Universal Robots PolyScope program: minipjoan.urp

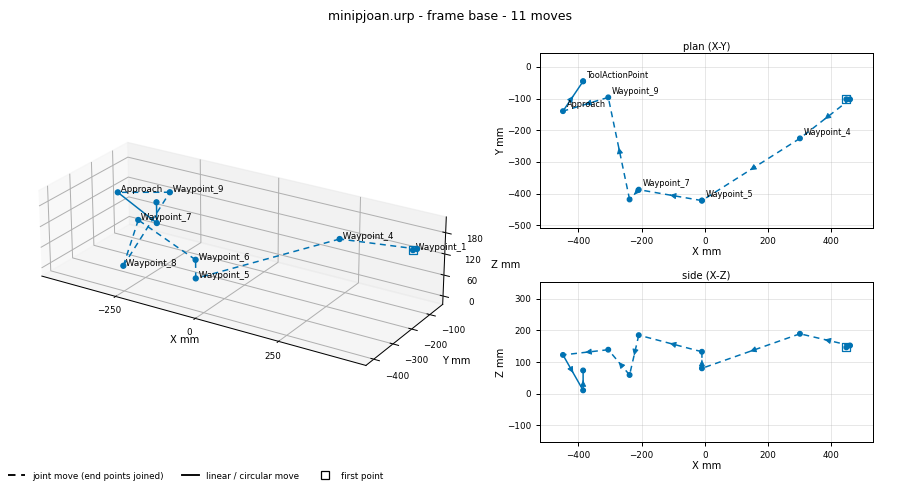
[picture p0: tool path of minipjoan.urp in frame base, 11 of 12 moves have a stored position in this frame; points joined in program order, loops and branches not executed]
Program minipjoan (installation=default directory=/programs createdIn=5.14.5 lastSavedIn=5.14.5 robotSerialNumber=20195300809)
Calibrated DH parameters: a=[-0.000085, -0.20076, -0.212369, 0.000121, -0.000118, 0]; d=[0.15185, -26.306375, 24.753047, 1.684739, 0.085386, 0.092088]; alpha=[1.572149, -0.00522, -0.011864, 1.571339, -1.571085, 0]; deltaTheta=[0, 0.599885, -0.513355, -0.086555, 0.000006, 0]
InitVariablesNode variables(variable(name=Pallet_1_cnt_1, expression=1), variable(name=Pallet_1_lct, expression=1), variable(name=Pallet_1_lno, expression=1), variable(name=Pallet_1_sep, expression=False), variable(name=Pallet_1_tct, expression=1))
Robot Program (runOnlyOnce=false)
  URCap Gripper Activate (Robotiq_Grippers, Robotiq Inc.) dataModel(ResetAndActivateKey=false)
  MoveJ speed 60 deg/s, acceleration 80 deg/s^2 (useActiveTCP=true) feature=Base
    Waypoint Waypoint_1: TCP in base x=447.267 y=-102.061 z=146.421 mm, rx=-2.205 ry=2.174 rz=-0.1317 rad; joints [4.81, -119.207, -49.648, -96.135, 87.137, 4.36] deg; TCP offset x=0 y=0 z=174 mm, rx=0 ry=0 rz=0 rad
  URCap Gripper (Robotiq_Grippers, Robotiq Inc.) dataModel(position=100.0, force=0.0, speed=0.0, positionInDouble=100.0, forceInDouble=0.0, speedInDouble=0.0, slaveIds=[9], blocking=true)
  MoveL speed 250 mm/s, acceleration 1200 mm/s^2 (useActiveTCP=true) feature=Base
    MoveDirectionNode (selectedDirection=ZMinus toolParams=0.05, 1.2)
      Until TOOL_CONTACT_DETECTION (allowActions=true retraction=0.005 decelerationAcceleration=3 decelerationAngularAcceleration=34.906585)
        URCap Gripper (Robotiq_Grippers, Robotiq Inc.) dataModel(position=0.0, force=0.0, speed=0.0, positionInDouble=0.0, forceInDouble=0.0, speedInDouble=0.0, slaveIds=[9], blocking=true)
        MoveL speed 250 mm/s, acceleration 1200 mm/s^2 (useActiveTCP=true) feature=Base
          Waypoint Waypoint_2 (Relative): relativeFromPosition TCP in base x=471.213 y=-99.416 z=63.282 mm, rx=-2.1249 ry=2.1283 rz=-0.2138 rad; joints [4.58, -119.887, -74.402, -64.902, 87.774, 4.609] deg; TCP in base x=479.804 y=-96.799 z=39.969 mm, rx=-2.142 ry=2.1284 rz=-0.2147 rad; joints [5.105, -123.73, -74.341, -61.658, 87.263, 4.605] deg
          URCap Gripper (Robotiq_Grippers, Robotiq Inc.) dataModel(position=58.431372549019606, force=0.0, speed=0.0, positionInDouble=58.431372549019606, forceInDouble=0.0, speedInDouble=0.0, slaveIds=[9], blocking=true)
          Waypoint Waypoint_3: TCP in base x=458.907 y=-102.285 z=152.325 mm, rx=-2.0281 ry=2.0188 rz=-0.3366 rad; joints [3.504, -105.987, -77.03, -66.932, 89.229, 3.326] deg
  MoveJ speed 60 deg/s, acceleration 80 deg/s^2 (useActiveTCP=true) feature=Base
    Waypoint Waypoint_4: TCP in base x=300.574 y=-225.676 z=189.373 mm, rx=-0.8393 ry=3.0246 rz=-0.1221 rad; joints [-13.828, -100.697, -62.451, -104.67, 85.518, 45.615] deg
    MoveJ speed 60 deg/s, acceleration 80 deg/s^2 (useActiveTCP=true) feature=Base
      Waypoint Waypoint_5: TCP in base x=-9.268 y=-422.356 z=80.192 mm, rx=-0.0596 ry=3.0948 rz=-0.085 rad; joints [-74.508, -112.122, -77.499, -76.664, 91.009, 13.565] deg
      URCap Gripper (Robotiq_Grippers, Robotiq Inc.) dataModel(position=0.0, force=0.0, speed=0.0, positionInDouble=0.0, forceInDouble=0.0, speedInDouble=0.0, slaveIds=[9], blocking=true)
      MoveJ speed 60 deg/s, acceleration 80 deg/s^2 (useActiveTCP=true) feature=Base
        Waypoint Waypoint_6: TCP in base x=-9.251 y=-422.355 z=132.542 mm, rx=-0.0597 ry=3.0948 rz=-0.085 rad; joints [-74.543, -111.435, -64.364, -90.485, 91.014, 13.69] deg
        Wait Sleep waitTime=8
    MoveJ speed 60 deg/s, acceleration 80 deg/s^2 (useActiveTCP=true) feature=Base
      Waypoint Waypoint_7: TCP in base x=-208.935 y=-387.816 z=185.052 mm, rx=0.0938 ry=-3.0517 rz=0.1155 rad; joints [44.36, -64.936, 47.012, -78.661, -91.033, -48.996] deg
      MoveJ speed 60 deg/s, acceleration 80 deg/s^2 (useActiveTCP=true) feature=Base
        Waypoint Waypoint_8: TCP in base x=-237.941 y=-418.796 z=59.161 mm, rx=0.0915 ry=-3.1228 rz=-0.0431 rad; joints [45.6, -46.032, 46.886, -90.484, -92.713, -47.784] deg
        URCap Gripper (Robotiq_Grippers, Robotiq Inc.) dataModel(position=58.03921568627451, force=0.0, speed=0.0, positionInDouble=58.03921568627451, forceInDouble=0.0, speedInDouble=0.0, slaveIds=[9], blocking=true)
      MoveJ speed 60 deg/s, acceleration 80 deg/s^2 (useActiveTCP=true) feature=Base
        Waypoint Waypoint_9: TCP in base x=-305.318 y=-96.059 z=139.035 mm, rx=-2.0283 ry=-2.295 rz=0.0831 rad; joints [-7.04, -97.483, 97.145, -95.102, -90.705, -13.988] deg
        URCap Palletizing (polyscope-pallet-impl, Universal Robots) dataModel(palletFeature=Base, isPalletizing=true, Variable(key=name, variable(name=Pallet_1)), Variable(key=globalCountingVariable, variable(name=Pallet_1_cnt_1, initializeExpression=1)), Variable(key=layerNumberVariable, variable(name=Pallet_1_lno, initializeExpression=1)), Variable(key=layerCountingVariable, variable(name=Pallet_1_lct, initializeExpression=1)), Variable(key=handleSeparatorVariable, variable(name=Pallet_1_sep, initializeExpression=False)), Variable(key=totalCountVariable, variable(name=Pallet_1_tct, initializeExpression=1)), Variable(key=referencePoint, variable(featureName=referencePoint)), Variable(key=separatorPoint, variable(featureName=separatorPoint)), Length(key=objectHeight value=0.04 unit=M)); state(isChildrenLocked=true)
          URCap Patterns (polyscope-pallet-impl, Universal Robots) state(isChildrenLocked=true)
            URCap Pattern (polyscope-pallet-impl, Universal Robots) dataModel(UUID=86fc2707-347a-4276-997c-d25539b2d56b, patternType=GRID, rows=3, columns=4, Variable(key=nameVariable, variable(name=Grid_Pattern_1))); state(isChildrenLocked=true)
              URCap Item (polyscope-pallet-impl, Universal Robots) dataModel(UUID=84c2eab7-4ccd-47c8-9968-c744c75cb5a4, patternType=GRID, index=0, calibrationDeltaTheta=[2.0871938292282843E-8, 0.5998849625986696, -0.513354759222901, -0.08655474087847535, 6.239817607139875E-6, -6.658617090343766E-8], calibrationA=[-8.52060452638757E-5, -0.2007601879611388, -0.2123691625519033, 1.2105607098011576E-4, -1.1833705743435544E-4, 0.0], calibrationD=[0.15184970286177432, -26.306374840159272, 24.75304670983349, 1.6847390881089916, 0.085385969004481, 0.09208826337351553], calibrationAlpha=[1.5721487795181908, -0.005219907129425837, -0.011864150755780208, 1.5713392161993658, -1.5710853432049288, 0.0], calibrationJointChecksum=[-1860213401, -1859864814, -1494669377, -1328152407, -1329437658, -1329056899], calibrationStatus=2, calibrationValidChecksum=true, baseToFeature=[0.0, 0.0, 0.0, 0.0, 0.0, 0.0], TCPOffset=[-4.9798563925285144E-8, -1.1903855710371225E-5, 0.17398545185544173, 3.862269624087422E-5, 1.2921357085209562E-5, -2.2884874203884517E-5], Variable(key=variable, variable(name=CornerItem_1)), JointPositions(key=jointpositions, JointPosition(key=[1], Angle(key=pos value=-0.188365 unit=RAD)), JointPosition(key=[2], Angle(key=pos value=-1.19048 unit=RAD)), JointPosition(key=[3], Angle(key=pos value=1.760904 unit=RAD)), JointPosition(key=[4], Angle(key=pos value=-2.274609 unit=RAD)), JointPosition(key=[5], Angle(key=pos value=-1.616725 unit=RAD)), JointPosition(key=[6], Angle(key=pos value=-0.207331 unit=RAD))))
              URCap Item (polyscope-pallet-impl, Universal Robots) dataModel(UUID=72bba91b-081b-49f2-b649-66cb13c50b99, patternType=GRID, index=1, calibrationDeltaTheta=[2.0871938292282843E-8, 0.5998849625986696, -0.513354759222901, -0.08655474087847535, 6.239817607139875E-6, -6.658617090343766E-8], calibrationA=[-8.52060452638757E-5, -0.2007601879611388, -0.2123691625519033, 1.2105607098011576E-4, -1.1833705743435544E-4, 0.0], calibrationD=[0.15184970286177432, -26.306374840159272, 24.75304670983349, 1.6847390881089916, 0.085385969004481, 0.09208826337351553], calibrationAlpha=[1.5721487795181908, -0.005219907129425837, -0.011864150755780208, 1.5713392161993658, -1.5710853432049288, 0.0], calibrationJointChecksum=[-1860213401, -1859864814, -1494669377, -1328152407, -1329437658, -1329056899], calibrationStatus=2, calibrationValidChecksum=true, baseToFeature=[0.0, 0.0, 0.0, 0.0, 0.0, 0.0], TCPOffset=[1.7947581433003235E-5, -3.939882102177439E-6, 0.17400140320939605, -8.22564695417386E-6, 3.537882574940382E-5, 3.057581507744186E-5], Variable(key=variable, variable(name=CornerItem_2)), JointPositions(key=jointpositions, JointPosition(key=[1], Angle(key=pos value=0.287634 unit=RAD)), JointPosition(key=[2], Angle(key=pos value=-0.966283 unit=RAD)), JointPosition(key=[3], Angle(key=pos value=1.377843 unit=RAD)), JointPosition(key=[4], Angle(key=pos value=-2.126769 unit=RAD)), JointPosition(key=[5], Angle(key=pos value=-1.625643 unit=RAD)), JointPosition(key=[6], Angle(key=pos value=0.264865 unit=RAD))))
              URCap Item (polyscope-pallet-impl, Universal Robots) dataModel(UUID=a3792030-abf1-4982-9561-2b57793ae55e, patternType=GRID, index=2, calibrationDeltaTheta=[2.0871938292282843E-8, 0.5998849625986696, -0.513354759222901, -0.08655474087847535, 6.239817607139875E-6, -6.658617090343766E-8], calibrationA=[-8.52060452638757E-5, -0.2007601879611388, -0.2123691625519033, 1.2105607098011576E-4, -1.1833705743435544E-4, 0.0], calibrationD=[0.15184970286177432, -26.306374840159272, 24.75304670983349, 1.6847390881089916, 0.085385969004481, 0.09208826337351553], calibrationAlpha=[1.5721487795181908, -0.005219907129425837, -0.011864150755780208, 1.5713392161993658, -1.5710853432049288, 0.0], calibrationJointChecksum=[-1860213401, -1859864814, -1494669377, -1328152407, -1329437658, -1329056899], calibrationStatus=2, calibrationValidChecksum=true, baseToFeature=[0.0, 0.0, 0.0, 0.0, 0.0, 0.0], TCPOffset=[2.0563843601384413E-5, -1.7894610874091832E-5, 0.1739782077066638, 5.339463614774784E-5, 5.4409430010765385E-5, 3.2483040918373374E-6], Variable(key=variable, variable(name=CornerItem_3)), JointPositions(key=jointpositions, JointPosition(key=[1], Angle(key=pos value=-0.160783 unit=RAD)), JointPosition(key=[2], Angle(key=pos value=-0.813561 unit=RAD)), JointPosition(key=[3], Angle(key=pos value=1.175602 unit=RAD)), JointPosition(key=[4], Angle(key=pos value=-2.219277 unit=RAD)), JointPosition(key=[5], Angle(key=pos value=-1.596708 unit=RAD)), JointPosition(key=[6], Angle(key=pos value=-0.11893 unit=RAD))))
              URCap Item (polyscope-pallet-impl, Universal Robots) dataModel(UUID=bd1f6cc1-746a-49c3-8aef-f84107da733c, patternType=GRID, index=3, calibrationDeltaTheta=[2.0871938292282843E-8, 0.5998849625986696, -0.513354759222901, -0.08655474087847535, 6.239817607139875E-6, -6.658617090343766E-8], calibrationA=[-8.52060452638757E-5, -0.2007601879611388, -0.2123691625519033, 1.2105607098011576E-4, -1.1833705743435544E-4, 0.0], calibrationD=[0.15184970286177432, -26.306374840159272, 24.75304670983349, 1.6847390881089916, 0.085385969004481, 0.09208826337351553], calibrationAlpha=[1.5721487795181908, -0.005219907129425837, -0.011864150755780208, 1.5713392161993658, -1.5710853432049288, 0.0], calibrationJointChecksum=[-1860213401, -1859864814, -1494669377, -1328152407, -1329437658, -1329056899], calibrationStatus=2, calibrationValidChecksum=true, baseToFeature=[0.0, 0.0, 0.0, 0.0, 0.0, 0.0], TCPOffset=[5.288007827730645E-7, 4.372061045532227E-6, 0.17401202246657863, -1.4752121198052903E-5, -5.497404895281797E-7, -2.6215338905465062E-6], Variable(key=variable, variable(name=CornerItem_4)), JointPositions(key=jointpositions, JointPosition(key=[1], Angle(key=pos value=0.216587 unit=RAD)), JointPosition(key=[2], Angle(key=pos value=-0.651099 unit=RAD)), JointPosition(key=[3], Angle(key=pos value=0.861928 unit=RAD)), JointPosition(key=[4], Angle(key=pos value=-2.089028 unit=RAD)), JointPosition(key=[5], Angle(key=pos value=-1.658829 unit=RAD)), JointPosition(key=[6], Angle(key=pos value=0.212513 unit=RAD))))
          URCap Layers (polyscope-pallet-impl, Universal Robots) dataModel(separators=[false], selectedPatterns=[86fc2707-347a-4276-997c-d25539b2d56b])
          URCap At Each Item (polyscope-pallet-impl, Universal Robots) dataModel(selectedPattern=86fc2707-347a-4276-997c-d25539b2d56b, selectedPosition=84c2eab7-4ccd-47c8-9968-c744c75cb5a4, Approach_calibrationDeltaTheta=[2.0871938292282843E-8, 0.5998849625986696, -0.513354759222901, -0.08655474087847535, 6.239817607139875E-6, -6.658617090343766E-8], Approach_calibrationA=[-8.52060452638757E-5, -0.2007601879611388, -0.2123691625519033, 1.2105607098011576E-4, -1.1833705743435544E-4, 0.0], Approach_calibrationD=[0.15184970286177432, -26.306374840159272, 24.75304670983349, 1.6847390881089916, 0.085385969004481, 0.09208826337351553], Approach_calibrationAlpha=[1.5721487795181908, -0.005219907129425837, -0.011864150755780208, 1.5713392161993658, -1.5710853432049288, 0.0], Approach_calibrationJointChecksum=[-1860213401, -1859864814, -1494669377, -1328152407, -1329437658, -1329056899], Approach_calibrationStatus=2, Approach_calibrationValidChecksum=true, Approach_baseToFeature=[0.0, 0.0, 0.0, 0.0, 0.0, 0.0], Approach_TCPOffset=[4.3887479497795034E-6, -2.1003613613068683E-5, 0.17399286414327153, 5.099101642133652E-5, -1.787022278136995E-5, 8.281297609357084E-6], Exit_calibrationDeltaTheta=[2.0871938292282843E-8, 0.5998849625986696, -0.513354759222901, -0.08655474087847535, 6.239817607139875E-6, -6.658617090343766E-8], Exit_calibrationA=[-8.52060452638757E-5, -0.2007601879611388, -0.2123691625519033, 1.2105607098011576E-4, -1.1833705743435544E-4, 0.0], Exit_calibrationD=[0.15184970286177432, -26.306374840159272, 24.75304670983349, 1.6847390881089916, 0.085385969004481, 0.09208826337351553], Exit_calibrationAlpha=[1.5721487795181908, -0.005219907129425837, -0.011864150755780208, 1.5713392161993658, -1.5710853432049288, 0.0], Exit_calibrationJointChecksum=[-1860213401, -1859864814, -1494669377, -1328152407, -1329437658, -1329056899], Exit_calibrationStatus=2, Exit_calibrationValidChecksum=true, Exit_baseToFeature=[0.0, 0.0, 0.0, 0.0, 0.0, 0.0], Exit_TCPOffset=[-1.3829321704010578E-6, 3.302622895939855E-6, 0.1740007596594772, -6.912230713125329E-6, -2.161785665733815E-5, 1.72877735477663E-5], currentWizardState=SHOW_DONE, Pose(key=refBaseToFeature, Position(key=posePosition, Length(key=X value=0 unit=M), Length(key=Y value=0 unit=M), Length(key=Z value=0 unit=M)), Rotation(key=poseRotation, Angle(key=RX value=0 unit=RAD), Angle(key=RY value=0 unit=RAD), Angle(key=RZ value=0 unit=RAD))), Pose(key=refPose, Position(key=posePosition, Length(key=X value=-0.386367 unit=M), Length(key=Y value=-0.044857 unit=M), Length(key=Z value=0.007745 unit=M)), Rotation(key=poseRotation, Angle(key=RX value=2.130527 unit=RAD), Angle(key=RY value=2.289871 unit=RAD), Angle(key=RZ value=-0.046413 unit=RAD))), JointPositions(key=Approach_jointpositions, JointPosition(key=[1], Angle(key=pos value=-0.253799 unit=RAD)), JointPosition(key=[2], Angle(key=pos value=-1.467465 unit=RAD)), JointPosition(key=[3], Angle(key=pos value=1.703907 unit=RAD)), JointPosition(key=[4], Angle(key=pos value=-1.940054 unit=RAD)), JointPosition(key=[5], Angle(key=pos value=-1.550823 unit=RAD)), JointPosition(key=[6], Angle(key=pos value=-0.278006 unit=RAD))), JointPositions(key=Exit_jointpositions, JointPosition(key=[1], Angle(key=pos value=-0.253518 unit=RAD)), JointPosition(key=[2], Angle(key=pos value=-1.450854 unit=RAD)), JointPosition(key=[3], Angle(key=pos value=1.673336 unit=RAD)), JointPosition(key=[4], Angle(key=pos value=-1.91882 unit=RAD)), JointPosition(key=[5], Angle(key=pos value=-1.550762 unit=RAD)), JointPosition(key=[6], Angle(key=pos value=-0.330343 unit=RAD))))
            URCap Generated Movements (polyscope-pallet-impl, Universal Robots) state(isChildrenLocked=true)
              MoveJ speed 60 deg/s, acceleration 80 deg/s^2 (useActiveTCP=true) feature=referencePoint
                Waypoint Approach: TCP in base x=-448.498 y=-139.667 z=122.58 mm, rx=-2.0744 ry=-2.0812 rz=0.3243 rad; joints [0.243, -70.586, 78.517, -114.353, -89.502, 0] deg; feature pose in base x=-386.367 y=-44.857 z=7.745 mm, rx=2.1305 ry=2.2899 rz=-0.0464 rad
              MoveL speed 250 mm/s, acceleration 1200 mm/s^2 (useActiveTCP=true) feature(featureName=referencePoint)
                Waypoint ToolActionPoint: TCP in base x=-384.793 y=-45.22 z=10.546 mm, rx=-2.1252 ry=-2.2993 rz=0.143 rad; joints [-16.512, -71.609, 103.51, -124.588, -86.188, -21.204] deg; feature pose in base x=-386.367 y=-44.857 z=7.745 mm, rx=2.1305 ry=2.2899 rz=-0.0464 rad
              Folder Tool action
                URCap Gripper (Robotiq_Grippers, Robotiq Inc.) dataModel(position=0.0, force=0.0, speed=0.0, positionInDouble=0.0, forceInDouble=0.0, speedInDouble=0.0, slaveIds=[9], blocking=true)
              MoveL speed 250 mm/s, acceleration 1200 mm/s^2 (useActiveTCP=true) feature(featureName=referencePoint)
                Waypoint Exit_1: TCP in base x=-384.778 y=-45.254 z=73.464 mm, rx=-2.1253 ry=-2.2994 rz=0.143 rad; joints [-16.556, -77.526, 92.92, -108.088, -86.265, -21.058] deg
Thread Thread_1 (runOnlyOnce=false)
  If digital_in[0]≟ True
    Set DigitalOutput pin=digital_out[0]; digitalValue=1
  Else 
    Set DigitalOutput pin=digital_out[0]; digitalValue=0
